// TIA Portal V16 export
// export: Created 2025-08-01T13:37:59.187325Z, ExportSetting WithDefaults, DisplayName Totally Integrated Automation Portal, DisplayVersion V16, DisplayName TIA Portal Version Control Interface, DisplayVersion V16, DisplayName TIA Portal Openness, DisplayVersion V16, DisplayName STEP 7 Professional, DisplayVersion V16, DisplayName STEP 7 Safety, DisplayVersion V16, DisplayName WinCC Advanced, DisplayVersion V16
FUNCTION_BLOCK "Delayed_Message_Function"   // FB2, FBD
TITLE = Delayed Message Function
VERSION : 0.1
// Functionblock For Delaying Message Function for example for filling an magazine or waiting for an signal. It is possible to adjust Time with the Dleay Time Message Input. The FlashTimer Time 1 & 2 ar for adjusting the flashing time of the ouput LED.
// stored: AutoNumber true, IsIECCheckEnabled false, UDAEnableTagReadback false
   VAR_INPUT
      "Override Message" : Bool;
      "Sensor Input 1" : Bool;
      "Sensor Input 2" : Bool := true;
      "Delay Time Message" : Time := T#1S_500MS;
      "FlashTimer Time 1" : Time := T#200ms;
      "FlashTimer Time 2" : Time := T#200ms;
   END_VAR
   VAR_OUTPUT
      "Output Signal" : Bool;
      "Output Signal Halt" : Bool;
      "ET Delayed Timer" : Time;
      "Output LED Flashing" : Bool;
   END_VAR
   VAR_TEMP
      "Internal Delayed Signal" : Bool;
   END_VAR
   VAR_TEMP   // added for the SCL form of the ladder/FBD networks
      _w1 : Bool;
   END_VAR
BEGIN

REGION Network 1: Delayed Signal to Outputs
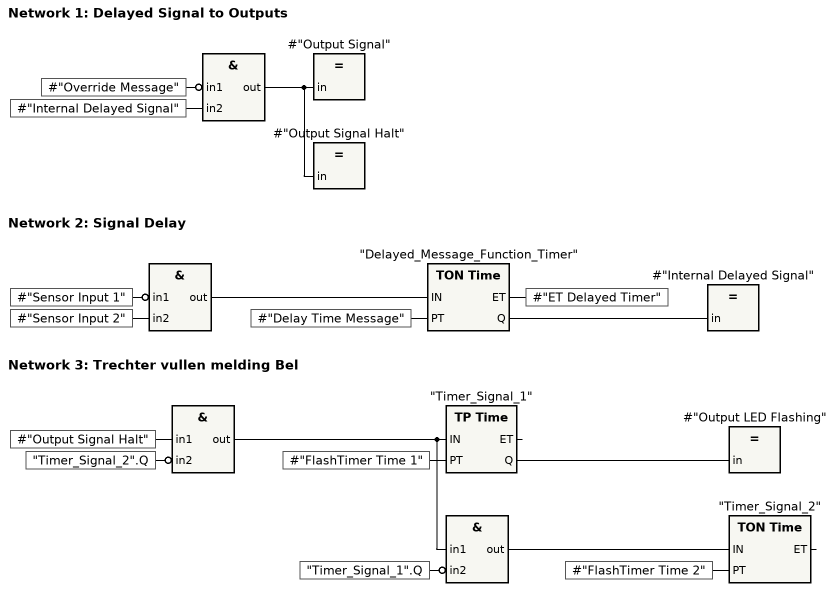
   #"Output Signal" := NOT #"Override Message" AND #"Internal Delayed Signal";
   #"Output Signal Halt" := #"Output Signal";
END_REGION

REGION Network 2: Signal Delay
   "Delayed_Message_Function_Timer".TON(IN := NOT #"Sensor Input 1" AND #"Sensor Input 2",
                           PT := #"Delay Time Message",
                           ET => #"ET Delayed Timer");
   #"Internal Delayed Signal" := "Delayed_Message_Function_Timer".Q;
END_REGION

REGION Network 3: Trechter vullen melding Bel
   #_w1 := #"Output Signal Halt" AND NOT "Timer_Signal_2".Q;
   "Timer_Signal_1".TP(IN := #_w1, PT := #"FlashTimer Time 1");
   #"Output LED Flashing" := "Timer_Signal_1".Q;
   "Timer_Signal_2".TON(IN := #_w1 AND NOT "Timer_Signal_1".Q, PT := #"FlashTimer Time 2");
END_REGION
END_FUNCTION_BLOCK
